// TIA Portal V16 export
// export: Created 2022-11-14T17:35:23.1759231Z, ExportSetting WithDefaults, DisplayName Totally Integrated Automation Portal, DisplayVersion V16, DisplayName TIA Portal Version Control Interface, DisplayVersion V16, DisplayName TIA Portal Openness, DisplayVersion V16, DisplayName STEP 7 Professional, DisplayVersion V16, DisplayName STEP 7 Safety, DisplayVersion V16, DisplayName WinCC Advanced, DisplayVersion V16
FUNCTION "FC18_ContrastCarriage" : Void   // FC18, LAD
TITLE = ContrastCarriage
{ S7_Optimized_Access := 'FALSE' }
VERSION : 0.1
// stored: AutoNumber false, IsIECCheckEnabled false, SetENOAutomatically false, UDAEnableTagReadback false
   VAR_TEMP   // added for the SCL form of the ladder/FBD networks
      _w1 : Bool;
   END_VAR
BEGIN

REGION Network 1: Timeout for welder contrast downward
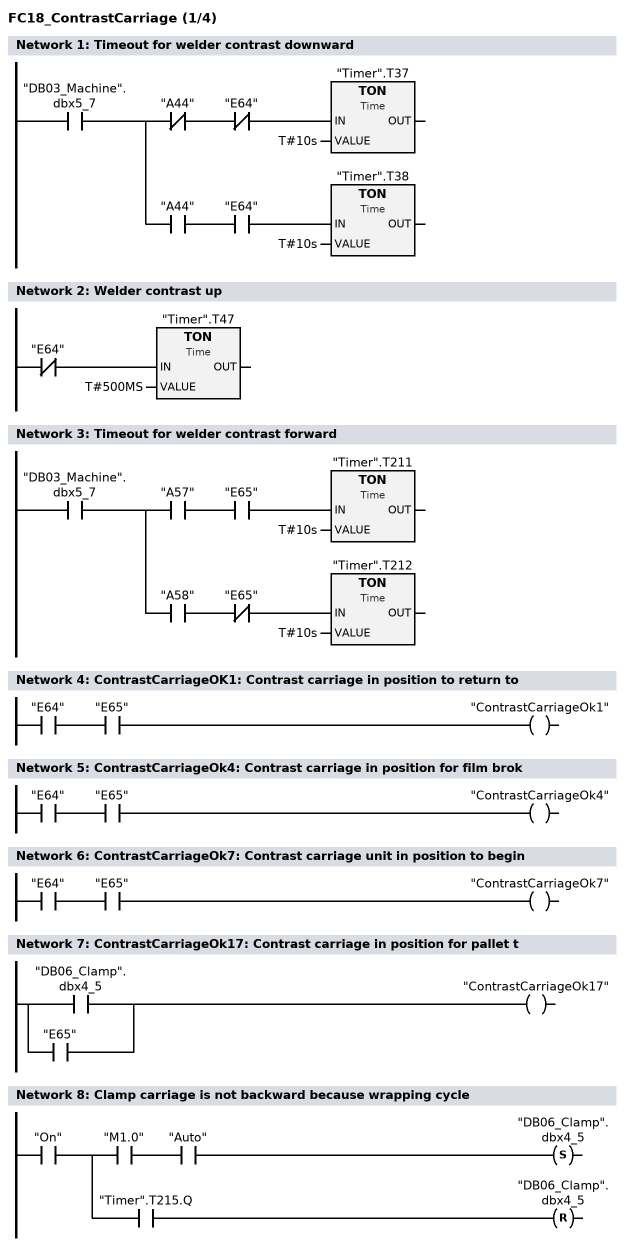
   "Timer".T37.TON(IN := "DB03_Machine".dbx5_7 AND NOT "A44" AND NOT "E64", PT := T#10s);   // TON coil
   "Timer".T38.TON(IN := "DB03_Machine".dbx5_7 AND "A44" AND "E64", PT := T#10s);   // TON coil
END_REGION

REGION Network 2: Welder contrast up
   "Timer".T47.TON(IN := NOT "E64", PT := T#500MS);   // TON coil
END_REGION

REGION Network 3: Timeout for welder contrast forward
   "Timer".T211.TON(IN := "DB03_Machine".dbx5_7 AND "A57" AND "E65", PT := T#10s);   // TON coil
   "Timer".T212.TON(IN := "DB03_Machine".dbx5_7 AND "A58" AND NOT "E65", PT := T#10s);   // TON coil
END_REGION

REGION Network 4: ContrastCarriageOK1: Contrast carriage in position to return to
   RUNG wire#powerrail
      Contact( "E64" )
      Contact( "E65" )
      Coil( "ContrastCarriageOk1" )
   END_RUNG
   // the same network as SCL:
   "ContrastCarriageOk1" := "E64" AND "E65";
END_REGION

REGION Network 5: ContrastCarriageOk4: Contrast carriage in position for film brok
   RUNG wire#powerrail
      Contact( "E64" )
      Contact( "E65" )
      Coil( "ContrastCarriageOk4" )
   END_RUNG
   // the same network as SCL:
   "ContrastCarriageOk4" := "E64" AND "E65";
END_REGION

REGION Network 6: ContrastCarriageOk7: Contrast carriage unit in position to begin
   RUNG wire#powerrail
      Contact( "E64" )
      Contact( "E65" )
      Coil( "ContrastCarriageOk7" )
   END_RUNG
   // the same network as SCL:
   "ContrastCarriageOk7" := "E64" AND "E65";
END_REGION

REGION Network 7: ContrastCarriageOk17: Contrast carriage in position for pallet t
   RUNG wire#powerrail
      Contact( "DB06_Clamp".dbx4_5 )
      wire#w1
      Coil( "ContrastCarriageOk17" )
   END_RUNG
   RUNG wire#powerrail
      Contact( "E65" )
   END_RUNG wire#w1
   // the same network as SCL:
   "ContrastCarriageOk17" := "DB06_Clamp".dbx4_5 OR "E65";
END_REGION

REGION Network 8: Clamp carriage is not backward because wrapping cycle
   RUNG wire#powerrail
      Contact( "On" )
      wire#w1
      Contact( "M1.0" )
      Contact( "Auto" )
      S_Coil( "DB06_Clamp".dbx4_5 )
   END_RUNG
   RUNG wire#w1
      Contact( "Timer".T215.Q )
      R_Coil( "DB06_Clamp".dbx4_5 )
   END_RUNG
   // the same network as SCL:
   IF "On" AND "M1.0" AND "Auto" THEN "DB06_Clamp".dbx4_5 := TRUE; END_IF;
   IF "On" AND "Timer".T215.Q THEN "DB06_Clamp".dbx4_5 := FALSE; END_IF;
END_REGION

REGION Network 9
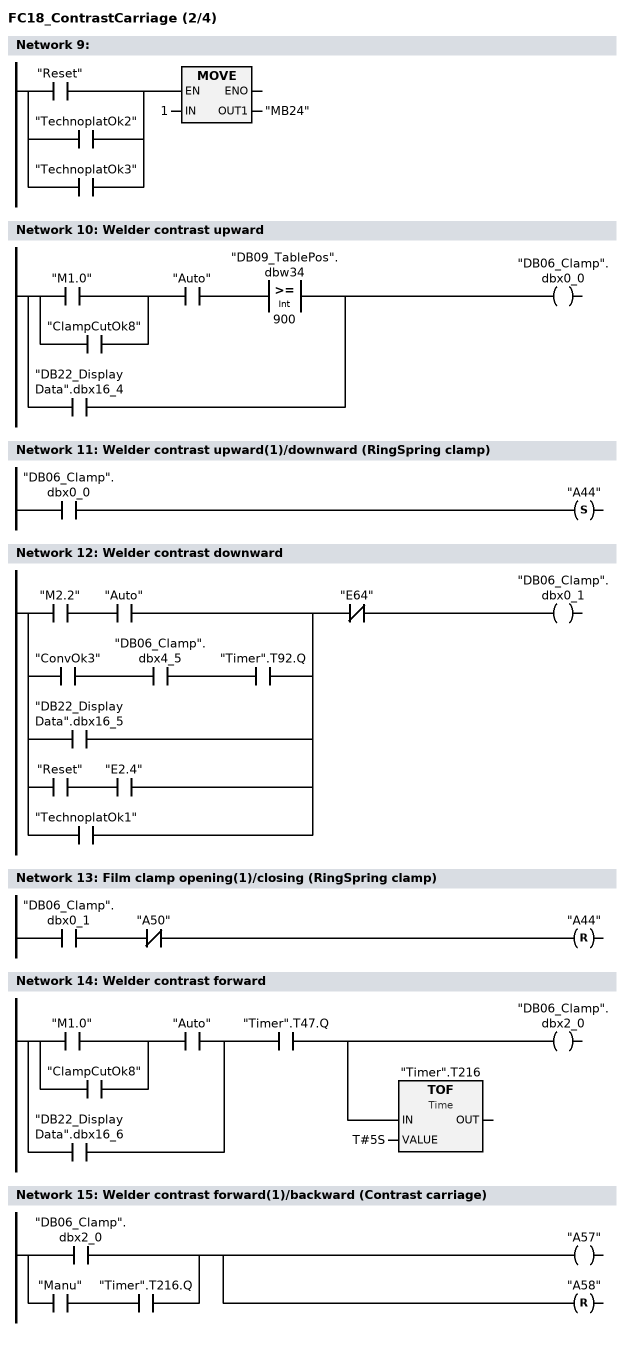
   RUNG wire#powerrail
      Contact( "Reset" )
      wire#w1
      { S7_GenerateENO := "TRUE" } Move(in := 1, out1 => "MB24")
   END_RUNG
   RUNG wire#powerrail
      Contact( "TechnoplatOk2" )
   END_RUNG wire#w1
   RUNG wire#powerrail
      Contact( "TechnoplatOk3" )
   END_RUNG wire#w1
   // the same network as SCL:
   IF "Reset" OR "TechnoplatOk2" OR "TechnoplatOk3" THEN "MB24" := 1; END_IF;
END_REGION

REGION Network 10: Welder contrast upward
   RUNG wire#powerrail
      Contact( "M1.0" )
      wire#w1
      Contact( "Auto" )
      { S7_Templates := "SrcType := Int" } GE_Contact(in1 := "DB09_TablePos".dbw34, in2 := 900)
      wire#w2
      Coil( "DB06_Clamp".dbx0_0 )
   END_RUNG
   RUNG wire#powerrail
      Contact( "ClampCutOk8" )
   END_RUNG wire#w1
   RUNG wire#powerrail
      Contact( "DB22_DisplayData".dbx16_4 )
   END_RUNG wire#w2
   // the same network as SCL:
   "DB06_Clamp".dbx0_0 := (("M1.0" OR "ClampCutOk8") AND "Auto" AND ("DB09_TablePos".dbw34 >= 900)) OR "DB22_DisplayData".dbx16_4;
END_REGION

REGION Network 11: Welder contrast upward(1)/downward (RingSpring clamp)
   RUNG wire#powerrail
      Contact( "DB06_Clamp".dbx0_0 )
      S_Coil( "A44" )
   END_RUNG
   // the same network as SCL:
   IF "DB06_Clamp".dbx0_0 THEN "A44" := TRUE; END_IF;
END_REGION

REGION Network 12: Welder contrast downward
   RUNG wire#powerrail
      Contact( "M2.2" )
      Contact( "Auto" )
      wire#w1
      I_Contact( "E64" )
      Coil( "DB06_Clamp".dbx0_1 )
   END_RUNG
   RUNG wire#powerrail
      Contact( "ConvOk3" )
      Contact( "DB06_Clamp".dbx4_5 )
      Contact( "Timer".T92.Q )
   END_RUNG wire#w1
   RUNG wire#powerrail
      Contact( "DB22_DisplayData".dbx16_5 )
   END_RUNG wire#w1
   RUNG wire#powerrail
      Contact( "Reset" )
      Contact( "E2.4" )
   END_RUNG wire#w1
   RUNG wire#powerrail
      Contact( "TechnoplatOk1" )
   END_RUNG wire#w1
   // the same network as SCL:
   "DB06_Clamp".dbx0_1 := (("M2.2" AND "Auto") OR ("ConvOk3" AND "DB06_Clamp".dbx4_5 AND "Timer".T92.Q) OR "DB22_DisplayData".dbx16_5 OR ("Reset" AND "E2.4") OR "TechnoplatOk1") AND NOT "E64";
END_REGION

REGION Network 13: Film clamp opening(1)/closing (RingSpring clamp)
   RUNG wire#powerrail
      Contact( "DB06_Clamp".dbx0_1 )
      I_Contact( "A50" )
      R_Coil( "A44" )
   END_RUNG
   // the same network as SCL:
   IF "DB06_Clamp".dbx0_1 AND NOT "A50" THEN "A44" := FALSE; END_IF;
END_REGION

REGION Network 14: Welder contrast forward
   "DB06_Clamp".dbx2_0 := ((("M1.0" OR "ClampCutOk8") AND "Auto") OR "DB22_DisplayData".dbx16_6) AND "Timer".T47.Q;
   "Timer".T216.TOF(IN := "DB06_Clamp".dbx2_0, PT := T#5S);   // TOF coil
END_REGION

REGION Network 15: Welder contrast forward(1)/backward (Contrast carriage)
   RUNG wire#powerrail
      Contact( "DB06_Clamp".dbx2_0 )
      wire#w1
      Coil( "A57" )
   END_RUNG
   RUNG wire#powerrail
      Contact( "Manu" )
      Contact( "Timer".T216.Q )
   END_RUNG wire#w1
   RUNG wire#w1
      R_Coil( "A58" )
   END_RUNG
   // the same network as SCL:
   "A57" := "DB06_Clamp".dbx2_0 OR ("Manu" AND "Timer".T216.Q);
   IF "A57" THEN "A58" := FALSE; END_IF;
END_REGION

REGION Network 16: Welder contrast backward
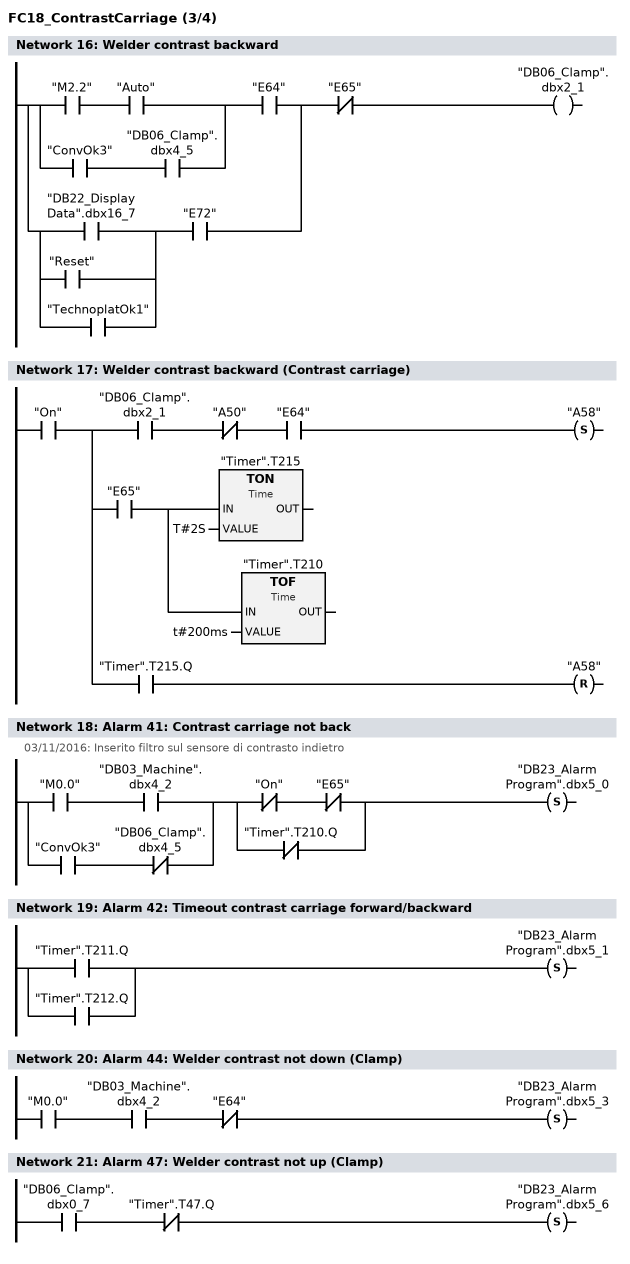
   RUNG wire#powerrail
      Contact( "M2.2" )
      Contact( "Auto" )
      wire#w1
      Contact( "E64" )
      wire#w2
      I_Contact( "E65" )
      Coil( "DB06_Clamp".dbx2_1 )
   END_RUNG
   RUNG wire#powerrail
      Contact( "ConvOk3" )
      Contact( "DB06_Clamp".dbx4_5 )
   END_RUNG wire#w1
   RUNG wire#powerrail
      Contact( "DB22_DisplayData".dbx16_7 )
      wire#w3
      Contact( "E72" )
   END_RUNG wire#w2
   RUNG wire#powerrail
      Contact( "Reset" )
   END_RUNG wire#w3
   RUNG wire#powerrail
      Contact( "TechnoplatOk1" )
   END_RUNG wire#w3
   // the same network as SCL:
   "DB06_Clamp".dbx2_1 := (((("M2.2" AND "Auto") OR ("ConvOk3" AND "DB06_Clamp".dbx4_5)) AND "E64") OR (("DB22_DisplayData".dbx16_7 OR "Reset" OR "TechnoplatOk1") AND "E72")) AND NOT "E65";
END_REGION

REGION Network 17: Welder contrast backward (Contrast carriage)
   IF "On" AND "DB06_Clamp".dbx2_1 AND NOT "A50" AND "E64" THEN "A58" := TRUE; END_IF;
   #_w1 := "On" AND "E65";
   "Timer".T215.TON(IN := #_w1, PT := T#2S);   // TON coil
   "Timer".T210.TOF(IN := #_w1, PT := t#200ms);   // TOF coil
   IF "On" AND "Timer".T215.Q THEN "A58" := FALSE; END_IF;
END_REGION

REGION Network 18: Alarm 41: Contrast carriage not back
   // 03/11/2016: Inserito filtro sul sensore di contrasto indietro
   RUNG wire#powerrail
      Contact( "M0.0" )
      Contact( "DB03_Machine".dbx4_2 )
      wire#w1
      I_Contact( "On" )
      I_Contact( "E65" )
      wire#w2
      S_Coil( "DB23_AlarmProgram".dbx5_0 )
   END_RUNG
   RUNG wire#powerrail
      Contact( "ConvOk3" )
      I_Contact( "DB06_Clamp".dbx4_5 )
   END_RUNG wire#w1
   RUNG wire#w1
      I_Contact( "Timer".T210.Q )
   END_RUNG wire#w2
   // the same network as SCL:
   IF (("M0.0" AND "DB03_Machine".dbx4_2) OR ("ConvOk3" AND NOT "DB06_Clamp".dbx4_5)) AND ((NOT "On" AND NOT "E65") OR NOT "Timer".T210.Q) THEN
       "DB23_AlarmProgram".dbx5_0 := TRUE;
   END_IF;
END_REGION

REGION Network 19: Alarm 42: Timeout contrast carriage forward/backward
   RUNG wire#powerrail
      Contact( "Timer".T211.Q )
      wire#w1
      S_Coil( "DB23_AlarmProgram".dbx5_1 )
   END_RUNG
   RUNG wire#powerrail
      Contact( "Timer".T212.Q )
   END_RUNG wire#w1
   // the same network as SCL:
   IF "Timer".T211.Q OR "Timer".T212.Q THEN "DB23_AlarmProgram".dbx5_1 := TRUE; END_IF;
END_REGION

REGION Network 20: Alarm 44: Welder contrast not down (Clamp)
   RUNG wire#powerrail
      Contact( "M0.0" )
      Contact( "DB03_Machine".dbx4_2 )
      I_Contact( "E64" )
      S_Coil( "DB23_AlarmProgram".dbx5_3 )
   END_RUNG
   // the same network as SCL:
   IF "M0.0" AND "DB03_Machine".dbx4_2 AND NOT "E64" THEN "DB23_AlarmProgram".dbx5_3 := TRUE; END_IF;
END_REGION

REGION Network 21: Alarm 47: Welder contrast not up (Clamp)
   RUNG wire#powerrail
      Contact( "DB06_Clamp".dbx0_7 )
      I_Contact( "Timer".T47.Q )
      S_Coil( "DB23_AlarmProgram".dbx5_6 )
   END_RUNG
   // the same network as SCL:
   IF "DB06_Clamp".dbx0_7 AND NOT "Timer".T47.Q THEN "DB23_AlarmProgram".dbx5_6 := TRUE; END_IF;
END_REGION

REGION Network 22: Alarm 50: Timeout for welder contrast upward/downward (Clamp)
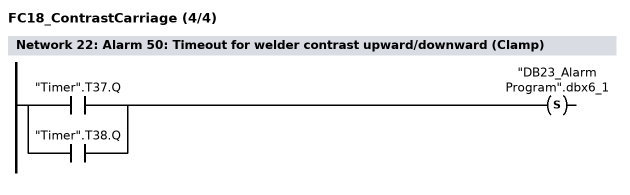
   RUNG wire#powerrail
      Contact( "Timer".T37.Q )
      wire#w1
      S_Coil( "DB23_AlarmProgram".dbx6_1 )
   END_RUNG
   RUNG wire#powerrail
      Contact( "Timer".T38.Q )
   END_RUNG wire#w1
   // the same network as SCL:
   IF "Timer".T37.Q OR "Timer".T38.Q THEN "DB23_AlarmProgram".dbx6_1 := TRUE; END_IF;
END_REGION
END_FUNCTION
